(* IEC 61131-3 sources: json/src, 3 files *)

(* ---- Constants.st ---- *)
NAMESPACE Simatic.Ax.Json
    TYPE
        Constants : Char (Strings := '"', Separator := ',') := Strings;
    END_TYPE
END_NAMESPACE

(* ---- JsonValueKind.st ---- *)
NAMESPACE Simatic.Ax.Json
    TYPE
        JsonValueKind : INT (_Array := 2, _False := 6, _Null := 7, _Number := 4, _Object := 1, _String := 3, _True := 5, _Undefined := 0) := _Undefined;
    END_TYPE
END_NAMESPACE

(* ---- IJsonObject.st ---- *)
NAMESPACE Simatic.Ax.Json
    INTERFACE IJsonObject
        METHOD ToString : STRING
        END_METHOD

        METHOD Serialize : BOOL
            VAR_INPUT
                t : Array[*] OF BYTE;
            END_VAR
        END_METHOD
    END_INTERFACE
END_NAMESPACE
